PROGRAM PRG_PUMP
VAR
	{attribute 'pytmc' := '
    pv: PTM:01
	'}
	PTM_01 :  FB_PTM_Pfeiffer;
	
	// They share the same serial port
	st_Pfeiffer_CTRL 			: ARRAY[1..20] OF ST_PfeifferControl;
	st_Pfeiffer_RBK 			: ARRAY[1..20] OF ST_PfeifferStatus;
	
	fb_PfeifferCom : FB_PFEIFFER_COM;
END_VAR



//Pfeiffer Turbo

(*Assign adresses to the pfeiffer controllers connected to this serial terminal*)
st_Pfeiffer_CTRL[1].iSerialAddress :=1;
st_Pfeiffer_CTRL[1].xEnableComm := TRUE;
	
(* Instanitate the Function block for serial communication with Pfeiffer*)	
fb_PfeifferCom(astPfeifferControl := st_Pfeiffer_CTRL,
			   astPfeifferStatus:= st_Pfeiffer_RBK,
				SerialRXBuffer:= E2_SerialRXBuffer,
				SerialTXBuffer:= E2_SerialTXBuffer);
				

(* Copy Status Pv's into the PTM structure*)
PTM_01.M_Serial_IO(st_Pfeiffer_CTRL[1],st_Pfeiffer_RBK[1]);

END_PROGRAM

(* stored: Version 1.1.0.1, ProductVersion 3.1.4024.2
   POU PRG_PUMP: Id {77bfa9ef-884a-40c8-8236-858350ca8c9b}, SpecialFunc None *)
